FUNCTION_BLOCK FB_Task EXTENDS FB_Object IMPLEMENTS I_Task, I_CyclicTask
VAR_INPUT
END_VAR
VAR_OUTPUT
END_VAR
VAR
    _eState:                E_TaskState;
    _eOldState:             E_TaskState;
    _nStartCounter:         UDINT := 0;
    fbExecutionTimer:       TON := (PT := TO_TIME(GVL_IntegerTypeBounds.DWORD_UPPER_BOUND));
    fbExecuteCallCtrl:      FB_InvocationControl;
END_VAR

METHOD Abort : I_TaskStatus
Abort := THIS^;

IF THIS^._eState = E_TaskState.Busy THEN
    THIS^.OnAbort();
    THIS^.Restore();
END_IF
END_METHOD

PROPERTY bBusy : BOOL
GET
bBusy := THIS^._eState = E_TaskState.Busy;
THIS^.CheckCyclicCall();
END_GET
END_PROPERTY

PROPERTY bDone : BOOL
GET
bDone := THIS^._eState = E_TaskState.Done;
THIS^.CheckCyclicCall();
END_GET
END_PROPERTY

PROPERTY bError : BOOL
GET
bError := THIS^._eState = E_TaskState.Error;
THIS^.CheckCyclicCall();
END_GET
END_PROPERTY

PROPERTY bReady : BOOL
GET
bReady := THIS^._eState = E_TaskState.Ready;
THIS^.CheckCyclicCall();
END_GET
END_PROPERTY

METHOD PRIVATE CheckCyclicCall
VAR_INST
    fbCallCtrl:             FB_InvocationControl;
END_VAR
fbCallCtrl.Track();

IF THIS^.eState = E_TaskState.Busy AND_THEN
    (THIS^.CyclicCallDropped()
        OR_ELSE (NOT THIS^.fbExecuteCallCtrl.bCalledCyclically AND_THEN fbCallCtrl.bNewInvocation)) THEN
    Tc2_System.ADSLOGSTR(
        msgCtrlMask := Tc2_System.ADSLOG_MSGTYPE_ERROR,
        msgFmtStr := 'Cyclic execution of is not done correctly for $'%s$'',
        strArg := THIS^.sPath);
END_IF
END_METHOD

METHOD PRIVATE CyclicCallDropped : BOOL
VAR_INST
    fbCyclicCallDropped:        F_TRIG;
END_VAR
fbCyclicCallDropped(CLK:= THIS^.fbExecuteCallCtrl.bCalledCyclically);

CyclicCallDropped := fbCyclicCallDropped.Q;
END_METHOD

METHOD DoneWhen : BOOL
VAR_INPUT
    bDone:          BOOL;
END_VAR
IF bDone AND_THEN THIS^._eState = E_TaskState.Busy THEN
    THIS^.SetState(E_TaskState.Done);
    THIS^.OnDone();
    DoneWhen := TRUE;
END_IF
END_METHOD

METHOD ErrorWhen : BOOL
VAR_INPUT
    bError:         BOOL;
END_VAR
IF bError AND_THEN THIS^._eState = E_TaskState.Busy THEN
    THIS^.SetState(E_TaskState.Error);
    THIS^.OnError();
    ErrorWhen := TRUE;
END_IF
END_METHOD

PROPERTY eState : E_TaskState
GET
eState := THIS^._eState;
END_GET
END_PROPERTY

METHOD PROTECTED Execute : BOOL
VAR_INPUT
END_VAR
THIS^.fbExecuteCallCtrl.Track();

IF THIS^._eState = E_TaskState.Error THEN
    THIS^.WhileError();
END_IF;

Execute := THIS^._eState = E_TaskState.Busy;

IF Execute THEN
    THIS^.fbExecutionTimer(IN := TRUE);
END_IF
END_METHOD

METHOD Invoke : I_TaskStatus
VAR_INST
    fbCallCtrl:         FB_InvocationControl;
END_VAR
fbCallCtrl.Track();

IF THIS^._eState = E_TaskState.Ready
    OR_ELSE ((THIS^._eState = E_TaskState.Done OR THIS^._eState = E_TaskState.Error) AND fbCallCtrl.bNewInvocation) THEN

    THIS^.SetState(E_TaskState.Busy);
    THIS^._nStartCounter := THIS^._nStartCounter + 1;
    THIS^.fbExecutionTimer(IN := FALSE);
    THIS^.OnStart();
END_IF

Invoke := THIS^;
END_METHOD

METHOD PROTECTED OnAbort
VAR_INPUT
END_VAR
END_METHOD

METHOD PROTECTED OnDone
VAR_INPUT
END_VAR
END_METHOD

METHOD PROTECTED OnError
VAR_INPUT
END_VAR
END_METHOD

METHOD PROTECTED OnStart
VAR_INPUT
END_VAR
END_METHOD

METHOD Restore : I_Restorable
THIS^.SetState(E_TaskState.Ready);
THIS^.fbExecutionTimer(IN := FALSE);

Restore := THIS^;
END_METHOD

METHOD Run
VAR_INPUT
END_VAR
END_METHOD

METHOD PRIVATE SetState
VAR_INPUT
    eNewState:          E_TaskState;
END_VAR
IF THIS^._eState <> eNewState THEN
    THIS^._eOldState := THIS^._eState;
    THIS^._eState := eNewState;
END_IF
END_METHOD

PROPERTY tElapsedTime : TIME
GET
tElapsedTime := fbExecutionTimer.ET;
END_GET
END_PROPERTY

METHOD PROTECTED WhileError
VAR_INPUT
END_VAR
END_METHOD

END_FUNCTION_BLOCK

(* stored: Version 1.1.0.1, ProductVersion 3.1.4024.12
   POU FB_Task: Id {f4d3bd7e-104a-4ada-800c-9a0a1d3ee958}, SpecialFunc None
   Folder Attributes: Id {0648b82d-b082-4066-b6d1-0d36afdd6bb0}
   Folder Cyclical: Id {a9d806fd-306e-428f-9745-b97ae33e30aa}
   Folder On Change: Id {7b54719e-317e-4661-bc93-15636e66b27e}
   Folder State Flow: Id {163a7df7-3015-49d9-b70e-8fd703683f52}
   Method Abort: Id {e29fef59-529d-4428-856d-a0423040ccee}
   Property bBusy: Id {adf293d6-cf35-403a-a60a-00c4af025de3}
   Get Get: Id {44e7a439-2fd7-49c3-bd5a-3f8064aeec64}
   Property bDone: Id {ab95c304-5686-42c0-a371-76fd93686585}
   Get Get: Id {d3893ab2-b012-405b-a4be-a71ce15f1199}
   Property bError: Id {5ae5e19f-ab56-4f17-8631-64e94506f4d0}
   Get Get: Id {a0def179-678c-49db-9708-1053c5bf7ed9}
   Property bReady: Id {483ad99a-a4ab-4cf1-ba7b-952c73d7eb27}
   Get Get: Id {aedb4938-68b4-4727-938a-ab71e6912d69}
   Method CheckCyclicCall: Id {b1a7e10b-f0c6-4efc-ab87-0b445b6ec704}
   Method CyclicCallDropped: Id {74e8aeb4-4e9c-4a50-82c8-677e7e19f117}
   Method DoneWhen: Id {15efd1b0-9d2e-4acd-85f4-d70243cc6597}
   Method ErrorWhen: Id {036c3caa-498b-4897-a6d5-ad8c4e8a1a30}
   Property eState: Id {c6d3fbdc-1f9b-42bd-a9c8-2d8c1aaa0363}
   Get Get: Id {4ec553bc-5f27-42d5-870f-192cfa04fd81}
   Method Execute: Id {2fa5e7f6-4779-4333-9846-d4ebf8c73074}
   Method Invoke: Id {7d291c31-c84c-4fd9-aa3e-9ccac03b239d}
   Method OnAbort: Id {5e42bc5c-9ca8-46d5-bc3a-561f8bb725c1}
   Method OnDone: Id {440178a0-fe57-41e7-a8b0-9dff8b47cefd}
   Method OnError: Id {72dbb8e6-5548-4ac3-b879-d778ada91edf}
   Method OnStart: Id {4ae4b885-beec-4640-9379-42cf5acf2fd5}
   Method Restore: Id {d3b160ff-5ff3-41c1-967f-4b834ff372cb}
   Method Run: Id {4a3124ce-aaa4-40fc-bfdd-6eec8224c877}
   Method SetState: Id {bc298fca-d865-460f-95bf-f2e5edbe4259}
   Property tElapsedTime: Id {4c0380ea-a1ab-48b4-95b2-7f8a3a65353e}
   Get Get: Id {5c36d2cd-cc24-4279-a355-f4e06a2f3f73}
   Method WhileError: Id {7cdf781c-f1d8-489d-bbf2-26d367973fff} *)
